(* IEC 61131-3 sources: IRIS-Project/LASAL CONTROL SOFTWARE/LasalProject_2025_09_12/Class/Manual_Step_Settings, 1 file *)

(* ---- Manual_Step_Settings.st ---- *)
(*!
<Class
	Name               = "Manual_Step_Settings"
	Revision           = "0.0"
	RealtimeTask       = "false"
	CyclicTask         = "true"
	DefCyclictime      = "500 ms"
	BackgroundTask     = "false"
	Sigmatek           = "false"
	OSInterface        = "false"
	HighPriority       = "false"
	Automatic          = "false"
	UpdateMode         = "Prescan"
	SharedCommandTable = "true"
	Objectsize         = "(900,1020)">
	<Channels>
		<Server Name="ClassSvr" Visualized="false" Initialize="false" WriteProtected="true" Retentive="false"/>
		<Server Name="M1_Exact_Step" Visualized="false" Initialize="false" WriteProtected="false" Retentive="false"/>
		<Server Name="M1_Moving_Step" Visualized="false" Initialize="false" WriteProtected="false" Retentive="false"/>
		<Server Name="M3_Exact_Step" Visualized="false" Initialize="false" WriteProtected="false" Retentive="false"/>
		<Server Name="M3_Moving_Step" Visualized="false" Initialize="false" WriteProtected="false" Retentive="false"/>
		<Server Name="M5_Charging_step_1" Visualized="false" Initialize="false" WriteProtected="false" Retentive="false"/>
		<Server Name="M5_Charging_step_2" Visualized="false" Initialize="false" WriteProtected="false" Retentive="false"/>
		<Server Name="M5_Charging_step_3" Visualized="false" Initialize="false" WriteProtected="false" Retentive="false"/>
		<Server Name="M5_Discharging_step_1" Visualized="false" Initialize="false" WriteProtected="false" Retentive="false"/>
		<Server Name="M5_Discharging_step_2" Visualized="false" Initialize="false" WriteProtected="false" Retentive="false"/>
		<Server Name="M5_Discharging_step_3" Visualized="false" Initialize="false" WriteProtected="false" Retentive="false"/>
		<Server Name="M5_Irradiation_step_1" Visualized="false" Initialize="false" WriteProtected="false" Retentive="false"/>
		<Server Name="M5_Irradiation_step_2" Visualized="false" Initialize="false" WriteProtected="false" Retentive="false"/>
		<Server Name="M5_Irradiation_step_3" Visualized="false" Initialize="false" WriteProtected="false" Retentive="false"/>
		<Client Name="c_M1_Exact_Step" Required="false" Internal="false"/>
		<Client Name="c_M1_Moving_Step" Required="false" Internal="false"/>
		<Client Name="c_M3_exact_Step" Required="true" Internal="false"/>
		<Client Name="c_M3_Moving_Step" Required="false" Internal="false"/>
		<Client Name="c_M5_Charging_Step_1" Required="true" Internal="false"/>
		<Client Name="c_M5_Charging_Step_2" Required="true" Internal="false"/>
		<Client Name="c_M5_Charging_Step_3" Required="true" Internal="false"/>
		<Client Name="c_M5_Discharging_step_1" Required="true" Internal="false"/>
		<Client Name="c_M5_Discharging_step_2" Required="true" Internal="false"/>
		<Client Name="c_M5_Discharging_step_3" Required="true" Internal="false"/>
		<Client Name="c_M5_Irradiation_Step_1" Required="true" Internal="false"/>
		<Client Name="c_M5_Irradiation_Step_2" Required="true" Internal="false"/>
		<Client Name="c_M5_Irradiation_step_3" Required="true" Internal="false"/>
	</Channels>
	<Separators>
		<Servers>
			<SepChn Position="3"/>
			<SepChn Position="6"/>
			<SepChn Position="10"/>
			<SepChn Position="14"/>
		</Servers>
		<Clients>
			<SepChn Position="2"/>
			<SepChn Position="5"/>
			<SepChn Position="9"/>
			<SepChn Position="13"/>
		</Clients>
	</Separators>
</Class>
*)
Manual_Step_Settings : CLASS
  //Servers:
	ClassSvr 	: SvrChCmd_DINT;
	M1_Moving_Step 	: SvrCh_DINT;
	M1_Exact_Step 	: SvrCh_DINT;
	M3_Moving_Step 	: SvrCh_DINT;
	M3_Exact_Step 	: SvrCh_DINT;
	M5_Charging_step_1 	: SvrCh_DINT;
	M5_Charging_step_2 	: SvrCh_DINT;
	M5_Charging_step_3 	: SvrCh_DINT;
	M5_Irradiation_step_1 	: SvrCh_DINT;
	M5_Irradiation_step_2 	: SvrCh_DINT;
	M5_Irradiation_step_3 	: SvrCh_DINT;
	M5_Discharging_step_1 	: SvrCh_DINT;
	M5_Discharging_step_2 	: SvrCh_DINT;
	M5_Discharging_step_3 	: SvrCh_DINT;
  //Clients:
	c_M1_Moving_Step 	: CltCh_DINT;
	c_M1_Exact_Step 	: CltCh_DINT;
	c_M3_Moving_Step 	: CltCh_DINT;
	c_M3_exact_Step 	: CltCh_DINT;
	c_M5_Charging_Step_1 	: CltCh_DINT;
	c_M5_Charging_Step_2 	: CltCh_DINT;
	c_M5_Charging_Step_3 	: CltCh_DINT;
	c_M5_Irradiation_Step_1 	: CltCh_DINT;
	c_M5_Irradiation_Step_2 	: CltCh_DINT;
	c_M5_Irradiation_step_3 	: CltCh_DINT;
	c_M5_Discharging_step_1 	: CltCh_DINT;
	c_M5_Discharging_step_2 	: CltCh_DINT;
	c_M5_Discharging_step_3 	: CltCh_DINT;
  //Variables:
		v_M1_MovingStep 	: DINT;
		v_M1_Exact_Step 	: DINT;
		v_M3_MovingStep 	: DINT;
		v_M3_Exact_Step 	: DINT;
		v_M5_Charging_step_1 	: DINT;
		v_M5_Charging_step_2 	: DINT;
		v_M5_Charging_step_3 	: DINT;
		v_M5_Irradiation_step_1 	: DINT;
		v_M5_Irradiation_step_2 	: DINT;
		v_M5_Irradiation_step_3 	: DINT;
		v_M5_Discahrging_step_1 	: DINT;
		v_M5_Discahrging_step_2 	: DINT;
		v_M5_Discahrging_step_3 	: DINT;
  //Functions:

	FUNCTION VIRTUAL GLOBAL Init;

	FUNCTION VIRTUAL GLOBAL CyWork
		VAR_INPUT
			EAX 	: UDINT;
		END_VAR
		VAR_OUTPUT
			state (EAX) 	: UDINT;
		END_VAR;

	FUNCTION VIRTUAL GLOBAL M1_Moving_Step::Read
		VAR_OUTPUT
			output (EAX) 	: DINT;
		END_VAR;

	FUNCTION VIRTUAL GLOBAL M1_Exact_Step::Read
		VAR_OUTPUT
			output (EAX) 	: DINT;
		END_VAR;

	FUNCTION VIRTUAL GLOBAL M3_Moving_Step::Read
		VAR_OUTPUT
			output (EAX) 	: DINT;
		END_VAR;

	FUNCTION VIRTUAL GLOBAL M3_Exact_Step::Read
		VAR_OUTPUT
			output (EAX) 	: DINT;
		END_VAR;

	FUNCTION VIRTUAL GLOBAL M5_Charging_step_1::Read
		VAR_OUTPUT
			output (EAX) 	: DINT;
		END_VAR;

	FUNCTION VIRTUAL GLOBAL M5_Charging_step_2::Read
		VAR_OUTPUT
			output (EAX) 	: DINT;
		END_VAR;

	FUNCTION VIRTUAL GLOBAL M5_Charging_step_3::Read
		VAR_OUTPUT
			output (EAX) 	: DINT;
		END_VAR;

	FUNCTION VIRTUAL GLOBAL M5_Irradiation_step_1::Read
		VAR_OUTPUT
			output (EAX) 	: DINT;
		END_VAR;

	FUNCTION VIRTUAL GLOBAL M5_Irradiation_step_2::Read
		VAR_OUTPUT
			output (EAX) 	: DINT;
		END_VAR;

	FUNCTION VIRTUAL GLOBAL M5_Irradiation_step_3::Read
		VAR_OUTPUT
			output (EAX) 	: DINT;
		END_VAR;

	FUNCTION VIRTUAL GLOBAL M5_Discharging_step_1::Read
		VAR_OUTPUT
			output (EAX) 	: DINT;
		END_VAR;

	FUNCTION VIRTUAL GLOBAL M5_Discharging_step_2::Read
		VAR_OUTPUT
			output (EAX) 	: DINT;
		END_VAR;

	FUNCTION VIRTUAL GLOBAL M5_Discharging_step_3::Read
		VAR_OUTPUT
			output (EAX) 	: DINT;
		END_VAR;
  //Tables:
	FUNCTION @STD
		VAR_OUTPUT
			ret_code	: CONFSTATES;
		END_VAR;
	FUNCTION GLOBAL TAB @CT_;
END_CLASS;

FUNCTION VIRTUAL GLOBAL Manual_Step_Settings::CyWork
	VAR_INPUT
		EAX 	: UDINT;
	END_VAR
	VAR_OUTPUT
		state (EAX) 	: UDINT;
	END_VAR

//READ FORM EPICS WITH MODBUS

if v_M1_MovingStep<>P_M1_C then
  v_M1_MovingStep:=M1_Moving_Step.Read();
end_if;

if v_M3_MovingStep<>P_M3_C then
  v_M3_MovingStep:=M3_Moving_Step.Read();
end_if;

v_M1_Exact_Step:=M1_Exact_Step.Read();
v_M3_Exact_Step:=M3_Exact_Step.Read();

if v_M5_Charging_step_1<>P1_M5 | v_M5_Charging_step_2<>P2_M5 | v_M5_Charging_step_3<>P3_M5 then
  v_M5_Charging_step_1:=M5_Charging_step_1.Read();
  v_M5_Charging_step_2:=M5_Charging_step_2.Read();
  v_M5_Charging_step_3:=M5_Charging_step_3.Read();
end_if;

if v_M5_Irradiation_step_1<>P1_M5_I | v_M5_Irradiation_step_2<>P2_M5_I | v_M5_Irradiation_step_3<>P3_M5_I then
  v_M5_Irradiation_step_1:=M5_Irradiation_step_1.Read();
  v_M5_Irradiation_step_2:=M5_Irradiation_step_2.Read();
  v_M5_Irradiation_step_3:=M5_Irradiation_step_3.Read();
end_if;

if v_M5_Discahrging_step_1<>P_M5_D | v_M5_Discahrging_step_2<>P_M5_D-OffsetDischarge | v_M5_Discahrging_step_3<>P_M5_D-2*OffsetDischarge then
  v_M5_Discahrging_step_1:=M5_Discharging_step_1.Read();
  v_M5_Discahrging_step_2:=M5_Discharging_step_2.Read();
  v_M5_Discahrging_step_3:=M5_Discharging_step_3.Read();
end_if;

//WRITE TO USE IN PLC

c_M1_Moving_Step.Write(input:=v_M1_MovingStep);
c_M1_Exact_Step.Write(input:=v_M1_Exact_Step);

c_M3_Moving_Step.Write(input:=v_M3_MovingStep);
c_M3_Exact_Step.Write(input:=v_M3_Exact_Step);

c_M5_Charging_step_1.Write(input:=v_M5_Charging_step_1);
c_M5_Charging_step_2.Write(input:=v_M5_Charging_step_2);
c_M5_Charging_step_3.Write(input:=v_M5_Charging_step_3);

c_M5_Irradiation_step_1.Write(input:=v_M5_Irradiation_step_1);
c_M5_Irradiation_step_2.Write(input:=v_M5_Irradiation_step_2);
c_M5_Irradiation_step_3.Write(input:=v_M5_Irradiation_step_3);

c_M5_Discharging_step_1.Write(input:=v_M5_Discahrging_step_1);
c_M5_Discharging_step_2.Write(input:=v_M5_Discahrging_step_2);
c_M5_Discharging_step_3.Write(input:=v_M5_Discahrging_step_3);

	state := READY;
END_FUNCTION

FUNCTION VIRTUAL GLOBAL Manual_Step_Settings::M5_Charging_step_1::Read
	VAR_OUTPUT
		output (EAX) 	: DINT;
	END_VAR

	output := M5_Charging_step_1;

END_FUNCTION

FUNCTION VIRTUAL GLOBAL Manual_Step_Settings::M5_Charging_step_2::Read
	VAR_OUTPUT
		output (EAX) 	: DINT;
	END_VAR

	output := M5_Charging_step_2;

END_FUNCTION

FUNCTION VIRTUAL GLOBAL Manual_Step_Settings::M5_Charging_step_3::Read
	VAR_OUTPUT
		output (EAX) 	: DINT;
	END_VAR

	output := M5_Charging_step_3;

END_FUNCTION

FUNCTION VIRTUAL GLOBAL Manual_Step_Settings::M5_Irradiation_step_1::Read
	VAR_OUTPUT
		output (EAX) 	: DINT;
	END_VAR

	output := M5_Irradiation_step_1;

END_FUNCTION

FUNCTION VIRTUAL GLOBAL Manual_Step_Settings::M5_Irradiation_step_2::Read
	VAR_OUTPUT
		output (EAX) 	: DINT;
	END_VAR

	output := M5_Irradiation_step_2;

END_FUNCTION

FUNCTION VIRTUAL GLOBAL Manual_Step_Settings::M5_Irradiation_step_3::Read
	VAR_OUTPUT
		output (EAX) 	: DINT;
	END_VAR

	output := M5_Irradiation_step_3;

END_FUNCTION

FUNCTION VIRTUAL GLOBAL Manual_Step_Settings::M5_Discharging_step_1::Read
	VAR_OUTPUT
		output (EAX) 	: DINT;
	END_VAR

	output := M5_Discharging_step_1;

END_FUNCTION

FUNCTION VIRTUAL GLOBAL Manual_Step_Settings::M5_Discharging_step_2::Read
	VAR_OUTPUT
		output (EAX) 	: DINT;
	END_VAR

	output := M5_Discharging_step_2;

END_FUNCTION

FUNCTION VIRTUAL GLOBAL Manual_Step_Settings::M5_Discharging_step_3::Read
	VAR_OUTPUT
		output (EAX) 	: DINT;
	END_VAR

	output := M5_Discharging_step_3;

END_FUNCTION

FUNCTION VIRTUAL GLOBAL Manual_Step_Settings::M1_Moving_Step::Read
	VAR_OUTPUT
		output (EAX) 	: DINT;
	END_VAR

	output := M1_Moving_Step;

END_FUNCTION

FUNCTION VIRTUAL GLOBAL Manual_Step_Settings::M1_Exact_Step::Read
	VAR_OUTPUT
		output (EAX) 	: DINT;
	END_VAR

	output := M1_Exact_Step;

END_FUNCTION

FUNCTION VIRTUAL GLOBAL Manual_Step_Settings::M3_Moving_Step::Read
	VAR_OUTPUT
		output (EAX) 	: DINT;
	END_VAR

	output := M3_Moving_Step;

END_FUNCTION

FUNCTION VIRTUAL GLOBAL Manual_Step_Settings::M3_Exact_Step::Read
	VAR_OUTPUT
		output (EAX) 	: DINT;
	END_VAR

	output := M3_Exact_Step;

END_FUNCTION

FUNCTION VIRTUAL GLOBAL Manual_Step_Settings::Init

v_M1_MovingStep:=P_M1_C;
v_M1_Exact_Step:=0;

v_M3_MovingStep:=P_M3_C;
v_M3_Exact_Step:=0;

v_M5_Charging_step_1:=P1_M5;
v_M5_Charging_step_2:=P2_M5;
v_M5_Charging_step_3:=P3_M5;

v_M5_Irradiation_step_1:=P1_M5_I;
v_M5_Irradiation_step_2:=P2_M5_I;
v_M5_Irradiation_step_3:=P3_M5_I;

v_M5_Discahrging_step_1:=P_M5_D;
v_M5_Discahrging_step_2:=P_M5_D-OffsetDischarge;
v_M5_Discahrging_step_3:=P_M5_D-2*OffsetDischarge;

END_FUNCTION
